FUNCTION_BLOCK FB_ContactorNonFB IMPLEMENTS I_ActivePowerNoFB
VAR
	sName 		: STRING;
	poCoil		: FB_DigitalOutput;
END_VAR

METHOD MR_PowerOFF : BOOL
VAR_INPUT
END_VAR
poCoil.Out := FALSE;
MR_PowerOFF := TRUE;
END_METHOD

METHOD MR_PowerON : BOOL
VAR_INPUT
END_VAR
poCoil.Out := TRUE;
MR_PowerON := TRUE;
END_METHOD

PROPERTY Name : STRING
GET
Name := sName;
END_GET
SET
sName := Name;
END_SET
END_PROPERTY

PROPERTY PowerOffIsCalled : bool
GET
PowerOffIsCalled := poCoil.Out=FALSE;
END_GET
END_PROPERTY

PROPERTY PowerOnIsCalled : bool
GET
PowerOnIsCalled := poCoil.Out=TRUE;
END_GET
END_PROPERTY

PROPERTY Ref_poCoil : reference to fb_digitalOutput
GET
ref_poCoil ref= poCoil;
END_GET
END_PROPERTY

END_FUNCTION_BLOCK

(* stored: Version 1.1.0.1, ProductVersion 3.1.4024.12
   POU FB_ContactorNonFB: Id {8055df9a-fcf2-4aab-8951-1daf8136d408}, SpecialFunc None
   Method MR_PowerOFF: Id {f586367f-63e8-4000-9264-0308e5e1e7c9}
   Method MR_PowerON: Id {c3e3ebf4-5abb-46b7-9be9-bbbcb5319997}
   Property Name: Id {467b226b-92ec-4530-a3d8-1fd1b2172635}
   Get Get: Id {042d11fd-4c6a-489f-896a-b1b64fbda2ed}
   Set Set: Id {a449f54f-f120-4f00-9cea-a86fffb5d374}
   Property PowerOffIsCalled: Id {f4d29c3a-e2e0-4255-bb91-f7f85b18af44}
   Get Get: Id {a32138f6-16f5-45e1-88d6-e1b9f9364882}
   Property PowerOnIsCalled: Id {b5a9fd27-9adb-442c-b74a-4e5f2de99305}
   Get Get: Id {19fd6cd3-c798-4dbe-a900-370b14c9c952}
   Property Ref_poCoil: Id {f448b09b-740d-4081-992d-9df83dad2ffa}
   Get Get: Id {7906f1d6-582f-4f12-89e8-0e51f0d8257c} *)
